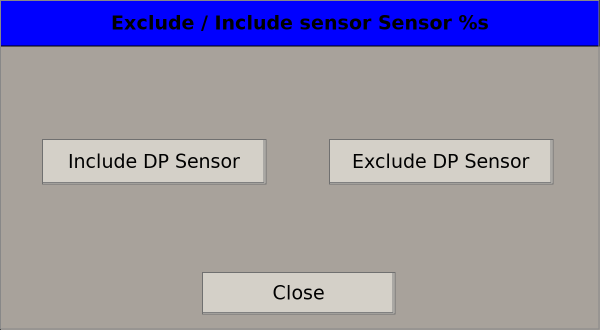
VISUALIZATION Dialog_DP_Field  // 600x330
VAR_IN_OUT
	sHeader: STRING;
	bSetPressIncluded: BOOL;
	bSetPressExcluded: BOOL;

END_VAR
    Rectangle (0,0 600x46), "Exclude / Include sensor Sensor %s", text variable: sHeader
    Button (42,139 224x45), "Include DP Sensor"
        OnMouseClick: execute { bSetPressIncluded:= TRUE; }
        OnMouseClick: CloseDialog Dialog=Dialog_CRAH, Result=OK, NumpadKeypadSet=True
    Button (329,139 224x45), "Exclude DP Sensor"
        OnMouseClick: execute { bSetPressExcluded:= TRUE; }
        OnMouseClick: CloseDialog Dialog=Dialog_DP_Field, Result=OK, NumpadKeypadSet=True
    Button (202,272 193x42), "Close"
        OnMouseClick: execute { bSetPressIncluded:= TRUE; }
        OnMouseClick: CloseDialog Dialog=Dialog_CRAH, Result=OK, NumpadKeypadSet=True
    Line (600,0) (600,330)
    Line (0,0) (0,330)
    Line (0,330) (600,330)
    Line (0,0) (600,0)
END_VISUALIZATION

(* stored: Version 1.1.0.1, ProductVersion 3.1.4024.12
   Visu Dialog_DP_Field: Id {9e8ba95d-2ee7-4016-bc64-8141ce4339c0} *)
